# EPICS StreamDevice protocol: tests/samples/patterns/documented/documented.proto
Terminator = CR LF;
getTemp { out "T?"; in "%f"; }
